// TIA Portal project "LONGHAI" (V15)

(* hardware
DEVICE "S7-1200 station_1"  S7-1200 Station
   slot 0: "Rack_0"  S7-1200 Rack  Rack  V1.0
   slot 1: "PLC_1"  CPU 1211C DC/DC/DC  6ES7 211-1AE40-0XB0  V4.2
*)

// ===== PLC "PLC_1"  CPU 1211C DC/DC/DC =====

VAR_GLOBAL   // PLC tag table "Default tag table"
   "Sensor" AT %I0.2 : Bool;
   "AUTO" AT %I0.3 : Bool;
   "MAN" AT %I0.4 : Bool;
   "Reset" AT %I0.5 : Bool;
   "Xilanh1" AT %Q0.0 : Bool;
   "Xilanh2" AT %Q0.1 : Bool;
   "Alarm_Auto" AT %Q0.2 : Bool;
   "Alarm_man" AT %Q0.3 : Bool;
   "SetPulse_Xilanh1_1" AT %MD5 : DInt;
   "WidthFulse" AT %MD50 : Time;
   "OnOff auto" AT %M2.0 : Bool;
   "OnOff man" AT %M2.1 : Bool;
   "ResetSW" AT %M2.2 : Bool;
   "KichReset" AT %M2.3 : Bool;
   "SetPulse_Xilanh1_2" AT %MD70 : DInt;
   "SetPulse_Xilanh2" AT %MD100 : Time;
   "sensor 2" AT %I0.1 : Bool;
   "System_Byte" AT %MB1 : Byte;
   "FirstScan" AT %M1.0 : Bool;
   "DiagStatusUpdate" AT %M1.1 : Bool;
   "AlwaysTRUE" AT %M1.2 : Bool;
   "AlwaysFALSE" AT %M1.3 : Bool;
   "Clock_Byte" AT %MB0 : Byte;
   "Clock_10Hz" AT %M0.0 : Bool;
   "Clock_5Hz" AT %M0.1 : Bool;
   "Clock_2.5Hz" AT %M0.2 : Bool;
   "Clock_2Hz" AT %M0.3 : Bool;
   "Clock_1.25Hz" AT %M0.4 : Bool;
   "Clock_1Hz" AT %M0.5 : Bool;
   "Clock_0.625Hz" AT %M0.6 : Bool;
   "Clock_0.5Hz" AT %M0.7 : Bool;
   "nho man" AT %M2.5 : Bool;
   "nho xl1" AT %M2.6 : Bool;
   "nho xl2" AT %M2.7 : Bool;
   "auto thung to" AT %M3.0 : Bool;
   "auto thung nho" AT %M3.1 : Bool;
END_VAR

// folder: System blocks/Program resources

DATA_BLOCK "IEC_Timer_0_DB_4"   // DB1
{ S7_Optimized_Access := 'TRUE' }
AUTHOR : Simatic
FAMILY : IEC
NAME : IEC_TMR
VERSION : 1.0
// stored: InstanceOfName IEC_TIMER
"IEC_TIMER"
BEGIN
END_DATA_BLOCK

DATA_BLOCK "IEC_Timer_0_DB"   // DB2
{ S7_Optimized_Access := 'TRUE' }
AUTHOR : Simatic
FAMILY : IEC
NAME : IEC_TMR
VERSION : 1.0
// stored: InstanceOfName IEC_TIMER
"IEC_TIMER"
BEGIN
END_DATA_BLOCK

DATA_BLOCK "IEC_Timer_0_DB_1"   // DB3
{ S7_Optimized_Access := 'TRUE' }
AUTHOR : Simatic
FAMILY : IEC
NAME : IEC_TMR
VERSION : 1.0
// stored: InstanceOfName IEC_TIMER
"IEC_TIMER"
BEGIN
END_DATA_BLOCK

DATA_BLOCK "IEC_Timer_0_DB_2"   // DB4
{ S7_Optimized_Access := 'TRUE' }
AUTHOR : Simatic
FAMILY : IEC
NAME : IEC_TMR
VERSION : 1.0
// stored: InstanceOfName IEC_TIMER
"IEC_TIMER"
BEGIN
END_DATA_BLOCK

DATA_BLOCK "IEC_Timer_0_DB_3"   // DB5
{ S7_Optimized_Access := 'TRUE' }
AUTHOR : Simatic
FAMILY : IEC
NAME : IEC_TMR
VERSION : 1.0
// stored: InstanceOfName IEC_TIMER
"IEC_TIMER"
BEGIN
END_DATA_BLOCK

DATA_BLOCK "IEC_Timer_0_DB_5"   // DB6
{ S7_Optimized_Access := 'TRUE' }
AUTHOR : Simatic
FAMILY : IEC
NAME : IEC_TMR
VERSION : 1.0
// stored: InstanceOfName IEC_TIMER
"IEC_TIMER"
BEGIN
END_DATA_BLOCK

DATA_BLOCK "IEC_Timer_0_DB_6"   // DB7
{ S7_Optimized_Access := 'TRUE' }
AUTHOR : Simatic
FAMILY : IEC
NAME : IEC_TMR
VERSION : 1.0
// stored: InstanceOfName IEC_TIMER
"IEC_TIMER"
BEGIN
END_DATA_BLOCK

// folder: (top level)

ORGANIZATION_BLOCK "Main"   // OB1, LAD, ProgramCycle
TITLE = "Main Program Sweep (Cycle)"
{ S7_Optimized_Access := 'TRUE' }
VERSION : 0.1
   VAR_INPUT
      Initial_Call : Bool;   // Initial call of this OB
      Remanence : Bool;   // =True, if remanent data are available
   END_VAR
   VAR_TEMP   // added for the SCL form of the ladder/FBD networks
      _w1 : Bool;
   END_VAR
BEGIN

REGION Network 1
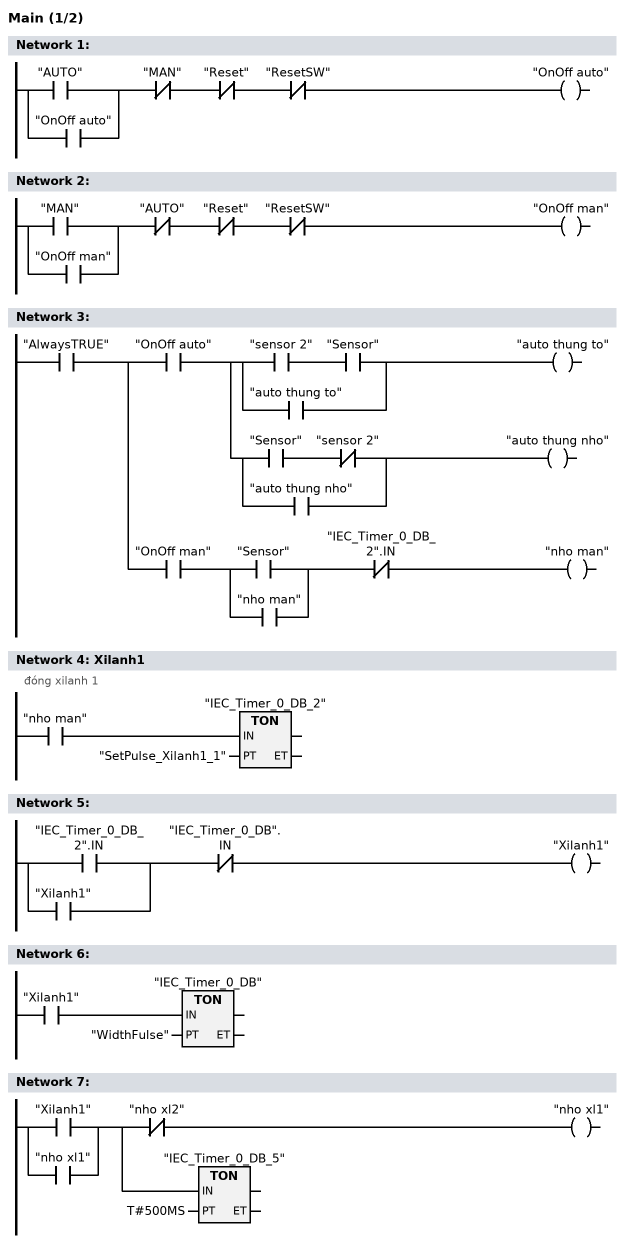
   RUNG wire#powerrail
      Contact( "AUTO" )
      wire#w1
      I_Contact( "MAN" )
      I_Contact( "Reset" )
      I_Contact( "ResetSW" )
      Coil( "OnOff auto" )
   END_RUNG
   RUNG wire#powerrail
      Contact( "OnOff auto" )
   END_RUNG wire#w1
   // the same network as SCL:
   "OnOff auto" := ("AUTO" OR "OnOff auto") AND NOT "MAN" AND NOT "Reset" AND NOT "ResetSW";
END_REGION

REGION Network 2
   RUNG wire#powerrail
      Contact( "MAN" )
      wire#w1
      I_Contact( "AUTO" )
      I_Contact( "Reset" )
      I_Contact( "ResetSW" )
      Coil( "OnOff man" )
   END_RUNG
   RUNG wire#powerrail
      Contact( "OnOff man" )
   END_RUNG wire#w1
   // the same network as SCL:
   "OnOff man" := ("MAN" OR "OnOff man") AND NOT "AUTO" AND NOT "Reset" AND NOT "ResetSW";
END_REGION

REGION Network 3
   RUNG wire#powerrail
      Contact( "AlwaysTRUE" )
      wire#w1
      Contact( "OnOff auto" )
      wire#w2
      Contact( "sensor 2" )
      Contact( "Sensor" )
      wire#w3
      Coil( "auto thung to" )
   END_RUNG
   RUNG wire#w2
      Contact( "auto thung to" )
   END_RUNG wire#w3
   RUNG wire#w2
      Contact( "Sensor" )
      I_Contact( "sensor 2" )
      wire#w4
      Coil( "auto thung nho" )
   END_RUNG
   RUNG wire#w2
      Contact( "auto thung nho" )
   END_RUNG wire#w4
   RUNG wire#w1
      Contact( "OnOff man" )
      wire#w5
      Contact( "Sensor" )
      wire#w6
      I_Contact( "IEC_Timer_0_DB_2".IN )
      Coil( "nho man" )
   END_RUNG
   RUNG wire#w5
      Contact( "nho man" )
   END_RUNG wire#w6
   // the same network as SCL:
   #_w1 := "AlwaysTRUE" AND "OnOff auto";
   "auto thung to" := #_w1 AND (("sensor 2" AND "Sensor") OR "auto thung to");
   "auto thung nho" := #_w1 AND (("Sensor" AND NOT "sensor 2") OR "auto thung nho");
   "nho man" := "AlwaysTRUE" AND "OnOff man" AND ("Sensor" OR "nho man") AND NOT "IEC_Timer_0_DB_2".IN;
END_REGION

REGION Network 4: Xilanh1
   // đóng xilanh 1
   "IEC_Timer_0_DB_2".TON(IN := "nho man", PT := "SetPulse_Xilanh1_1");
END_REGION

REGION Network 5
   RUNG wire#powerrail
      Contact( "IEC_Timer_0_DB_2".IN )
      wire#w1
      I_Contact( "IEC_Timer_0_DB".IN )
      Coil( "Xilanh1" )
   END_RUNG
   RUNG wire#powerrail
      Contact( "Xilanh1" )
   END_RUNG wire#w1
   // the same network as SCL:
   "Xilanh1" := ("IEC_Timer_0_DB_2".IN OR "Xilanh1") AND NOT "IEC_Timer_0_DB".IN;
END_REGION

REGION Network 6
   "IEC_Timer_0_DB".TON(IN := "Xilanh1", PT := "WidthFulse");
END_REGION

REGION Network 7
   #_w1 := "Xilanh1" OR "nho xl1";
   "nho xl1" := #_w1 AND NOT "nho xl2";
   "IEC_Timer_0_DB_5".TON(IN := #_w1, PT := T#500MS);
END_REGION

REGION Network 8
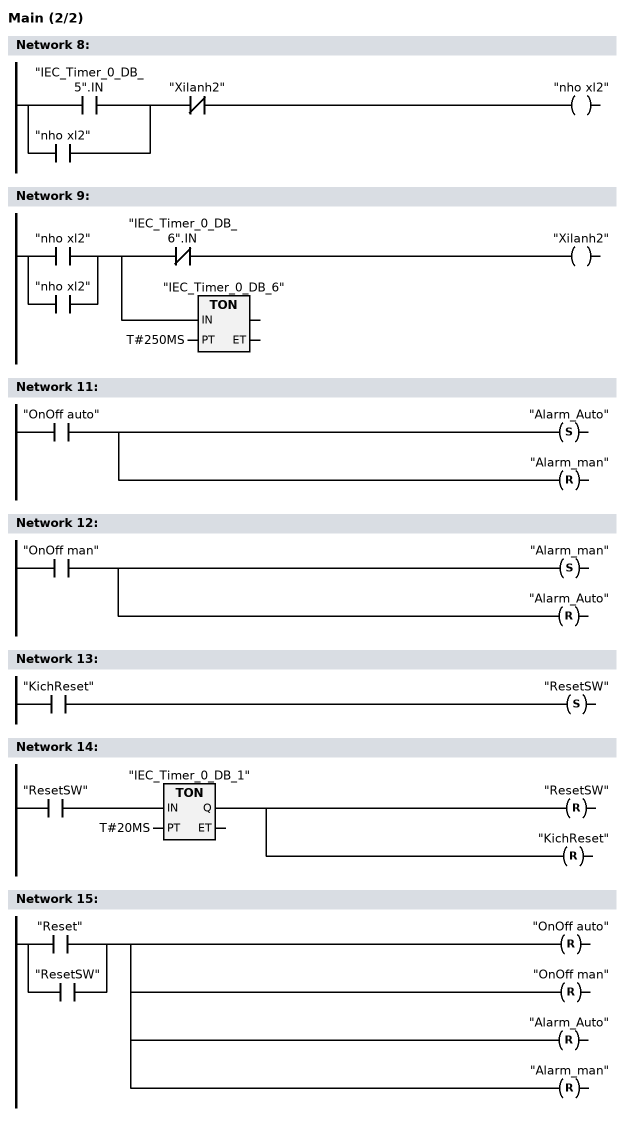
   RUNG wire#powerrail
      Contact( "IEC_Timer_0_DB_5".IN )
      wire#w1
      I_Contact( "Xilanh2" )
      Coil( "nho xl2" )
   END_RUNG
   RUNG wire#powerrail
      Contact( "nho xl2" )
   END_RUNG wire#w1
   // the same network as SCL:
   "nho xl2" := ("IEC_Timer_0_DB_5".IN OR "nho xl2") AND NOT "Xilanh2";
END_REGION

REGION Network 9
   #_w1 := "nho xl2" OR "nho xl2";
   "Xilanh2" := #_w1 AND NOT "IEC_Timer_0_DB_6".IN;
   "IEC_Timer_0_DB_6".TON(IN := #_w1, PT := T#250MS);
END_REGION

REGION Network 11
   RUNG wire#powerrail
      Contact( "OnOff auto" )
      wire#w1
      S_Coil( "Alarm_Auto" )
   END_RUNG
   RUNG wire#w1
      R_Coil( "Alarm_man" )
   END_RUNG
   // the same network as SCL:
   IF "OnOff auto" THEN
       "Alarm_Auto" := TRUE;
       "Alarm_man" := FALSE;
   END_IF;
END_REGION

REGION Network 12
   RUNG wire#powerrail
      Contact( "OnOff man" )
      wire#w1
      S_Coil( "Alarm_man" )
   END_RUNG
   RUNG wire#w1
      R_Coil( "Alarm_Auto" )
   END_RUNG
   // the same network as SCL:
   IF "OnOff man" THEN
       "Alarm_man" := TRUE;
       "Alarm_Auto" := FALSE;
   END_IF;
END_REGION

REGION Network 13
   RUNG wire#powerrail
      Contact( "KichReset" )
      S_Coil( "ResetSW" )
   END_RUNG
   // the same network as SCL:
   IF "KichReset" THEN "ResetSW" := TRUE; END_IF;
END_REGION

REGION Network 14
   "IEC_Timer_0_DB_1".TON(IN := "ResetSW", PT := T#20MS);
   IF "IEC_Timer_0_DB_1".Q THEN
       "ResetSW" := FALSE;
       "KichReset" := FALSE;
   END_IF;
END_REGION

REGION Network 15
   RUNG wire#powerrail
      Contact( "Reset" )
      wire#w1
      R_Coil( "OnOff auto" )
   END_RUNG
   RUNG wire#powerrail
      Contact( "ResetSW" )
   END_RUNG wire#w1
   RUNG wire#w1
      R_Coil( "OnOff man" )
   END_RUNG
   RUNG wire#w1
      R_Coil( "Alarm_Auto" )
   END_RUNG
   RUNG wire#w1
      R_Coil( "Alarm_man" )
   END_RUNG
   // the same network as SCL:
   IF "Reset" OR "ResetSW" THEN
       "OnOff auto" := FALSE;
       "OnOff man" := FALSE;
       "Alarm_Auto" := FALSE;
       "Alarm_man" := FALSE;
   END_IF;
END_REGION
END_ORGANIZATION_BLOCK